(*
============================================================
ST_MqttConfig
============================================================
PURPOSE
  MQTT broker connection and topic configuration.
  Populated from GVL_Config defaults on startup.
  Operator can override all fields from the HMI MQTT-Config
  panel, then press "Apply & Reconnect" to activate changes.

NOTES
  • Changing any field requires pressing Apply (triggers bApplyConfig
    rising edge in FB_MqttManager) to reconnect with new settings.
  • Use TLS (bUseTls = TRUE, nPort = 8883) for production deployments.
  • Credentials are NOT stored in persistent memory — they must be
    re-entered after a cold restart unless the HMI retains them.
============================================================
*)
TYPE ST_MqttConfig :
STRUCT
    (* ── Broker Connection ──────────────────────────────────── *)
    sBrokerAddress      : STRING(255) := 'imsiot.aws.thinger.io';   (* IP or hostname of MQTT broker     *)
    nPort               : UINT        := 1883;              (* 1883 = plain, 8883 = TLS/SSL      *)
    sClientId           : STRING(64)  := 'Beckhoff'; (* Must be unique per broker   *)
    sUsername           : STRING(64)  := 'ims_iot';                (* Leave empty if no auth required   *)
    sPassword           : STRING(64)  := '123456789';                (* Leave empty if no auth required   *)
    bUseTls             : BOOL        := FALSE;             (* TRUE enables TLS/SSL connection   *)

    (* ── Topic Configuration ────────────────────────────────── *)
    sTopicPrefix        : STRING(64)  := 'irrigation';      (* Base prefix for all topics        *)
    (* Publish topic  : <prefix>/status                                                           *)
    (* Subscribe topic: <prefix>/command                                                          *)
    sMainTopic          : STRING(128) := 'irrigation/status';   (* Full publish topic            *)
    SubscribeTopic      : STRING(128) := 'irrigation/command';  (* Full subscribe topic          *)

    (* ── Timing ─────────────────────────────────────────────── *)
    tStatusPublishInterval : TIME := T#5M;                  (* Cyclic publish interval (5 min)   *)
    tReconnectDelay        : TIME := T#30S;                 (* Back-off delay between retries    *)

    (* ── Runtime Control ────────────────────────────────────── *)
    bUseStatusPublish   : BOOL := TRUE;                     (* TRUE = publish status cyclically  *)
    bApplyConfig        : BOOL;                             (* Rising edge: reconnect with new cfg*)
END_STRUCT
END_TYPE

(* stored: Version 1.1.0.1, ProductVersion 3.1.4026.18
   DUT ST_MqttConfig: Id {0d23f381-9828-49b6-8416-3eaade8f2f19} *)
